// TIA Portal V16 export
// export: Created 2022-09-01T13:36:54.4748311Z, ExportSetting WithDefaults, DisplayName Totally Integrated Automation Portal, DisplayVersion V16, DisplayName TIA Portal Version Control Interface, DisplayVersion V16, DisplayName TIA Portal Openness, DisplayVersion V16, DisplayName STEP 7 Professional, DisplayVersion V16, DisplayName STEP 7 Safety, DisplayVersion V16, DisplayName WinCC Advanced, DisplayVersion V16
FUNCTION "Alarme_XV102" : Void   // FC24, LAD
{ S7_Optimized_Access := 'TRUE' }
VERSION : 0.1
// stored: AutoNumber true, IsIECCheckEnabled false, SetENOAutomatically false, UDAEnableTagReadback false
BEGIN

REGION Network 1: XV102 a abrir
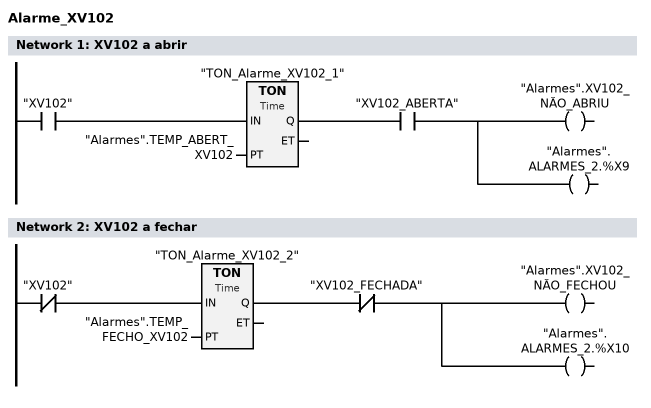
   RUNG wire#powerrail
      Contact( "XV102" )
      { S7_Templates := "time_type := Time" } "TON_Alarme_XV102_1".TON(pt := "Alarmes".TEMP_ABERT_XV102, et =>)
      Contact( "XV102_ABERTA" )
      wire#w1
      Coil( "Alarmes".XV102_NÃO_ABRIU )
   END_RUNG
   RUNG wire#w1
      Coil( "Alarmes".ALARMES_2.%X9 )
   END_RUNG
   // the same network as SCL:
   "TON_Alarme_XV102_1".TON(IN := "XV102", PT := "Alarmes".TEMP_ABERT_XV102);
   "Alarmes".XV102_NÃO_ABRIU := "TON_Alarme_XV102_1".Q AND "XV102_ABERTA";
   "Alarmes".ALARMES_2.%X9 := "Alarmes".XV102_NÃO_ABRIU;
END_REGION

REGION Network 2: XV102 a fechar
   RUNG wire#powerrail
      I_Contact( "XV102" )
      { S7_Templates := "time_type := Time" } "TON_Alarme_XV102_2".TON(pt := "Alarmes".TEMP_FECHO_XV102, et =>)
      I_Contact( "XV102_FECHADA" )
      wire#w1
      Coil( "Alarmes".XV102_NÃO_FECHOU )
   END_RUNG
   RUNG wire#w1
      Coil( "Alarmes".ALARMES_2.%X10 )
   END_RUNG
   // the same network as SCL:
   "TON_Alarme_XV102_2".TON(IN := NOT "XV102", PT := "Alarmes".TEMP_FECHO_XV102);
   "Alarmes".XV102_NÃO_FECHOU := "TON_Alarme_XV102_2".Q AND NOT "XV102_FECHADA";
   "Alarmes".ALARMES_2.%X10 := "Alarmes".XV102_NÃO_FECHOU;
END_REGION
END_FUNCTION
